TYPE Motion_PlcToHmi :
STRUCT
	actPos				: LREAL;
	actVelo				: LREAL;
	setPos				: LREAL; 
	setVelo 			: LREAL; 
	controller_override : LREAL;
	isDisabled 			: BOOL;
	isFwDisabled 		: BOOL;
	isBwDisabled 		: BOOL;
	isCalibrated		: BOOL;
	hasJob				: BOOL;
	isNotMoving 		: BOOL;
	isPositiveDirection : BOOL;
	isNegativeDirection : BOOL;            
    isInTarget 			: BOOL;            
    isInRange 			: BOOL;            
END_STRUCT
END_TYPE

(* stored: Version 1.1.0.1, ProductVersion 3.1.0.36
   DUT Motion_PlcToHmi: Id {1da300d1-f238-4497-b81a-36eb9fe7f711} *)
